// TIA Portal V21 export
DATA_BLOCK "GasBlanketing"   // DB308
AUTHOR : PRECISE
FAMILY : PRECISE
// stored: AutoNumber false, InstanceOfName FB304, InstanceOfType FB
"FB304"
   // VAR_INPUT
   //    Enable : Bool;
   //    Disable : Bool;
   //    Fault : Bool;
   //    SecPulse : Bool;
   //    AlwaysTrue : Bool;
   //    StartConfirmationPopupSel : Bool;
   //    EndConfirmationPopupSel : Bool;
   //    BlanketingModeSel : Int;
   //    BlanketingTimebaseSel : Bool;
   //    GasSel : Int;
   //    SetPressure : Real := 1.2;
   //    BlanketingTimeMin : Int;
   //    BlanketingTimeSec : Int;
   //    ActualPressure : Real;
   //    DelaytoOpenGasIn : Int;
   //    PressureTol : Real;
   // END_VAR
   // VAR_OUTPUT
   //    AirValve : Bool;
   //    N2Valve : Bool;
   //    BlanketingLineValves : Bool;
   //    StartConfirmationPopup : Bool;
   //    EndConfirmationPopup : Bool;
   //    BlanketingTimeMinPV : DInt;
   //    BlanketingTimeSecPV : DInt;
   //    PrintTrigger : Bool;
   //    PrintWord : Int;
   //    PrintStatus : String[50];
   // END_VAR
   // VAR_IN_OUT
   //    Start : Bool;
   //    Stop : Bool;
   //    Reset : Bool;
   //    StartConfirmationAck : Bool;
   //    EndConfirmationAck : Bool;
   //    SpareBtn1 : Bool;
   //    SpareBtn2 : Bool;
   //    SpareBtn3 : Bool;
   //    Running : Bool;
   //    Selected : Bool;
   //    Paused : Bool;
   //    StartConfirmationPopupTemp : Bool;
   //    EndConfirmationPopupTemp : Bool;
   //    BlanketingStarted : Bool;
   //    BlanketingOver : Bool;
   //    BlanketingTimerRunning : Bool;
   //    PressureTolNeg : Real;
   // END_VAR
   // VAR
   //    ValveOnDelayPV : Int;
   //    ValveOffDelayPV : Int;
   //    PrintTriggerTemp : Bool;
   //    RE1 : Bool;
   //    RE2 : Bool;
   //    RE3 : Bool;
   //    RE4 : Bool;
   //    RE5 : Bool;
   //    RE6 : Bool;
   //    RE7 : Bool;
   //    BlanketingTimer { S7_SetPoint := 'True'} : "FB101";
   //    PrintTriggerResetTimer { S7_SetPoint := 'True'} : TON_TIME;
   //    BtnResetTimer { S7_SetPoint := 'True'} : TON_TIME;
   // END_VAR
BEGIN
END_DATA_BLOCK
